FUNCTION_BLOCK FB_Status
VAR_INPUT
	eMode 	: E_Mode;
	fTime	: LREAL;
	bFault 	: BOOL;
END_VAR
VAR_OUTPUT
	eStatus : E_Status := E_Status.Checking;
END_VAR
VAR
	bRunning : BOOL;
END_VAR

IF fTime > 2.0 THEN
	bRunning := TRUE;
ELSE
	bRunning := FALSE;	
END_IF


CASE eStatus OF 
	E_Status.Checking:
		IF bFault THEN
			eStatus := E_Status.Fault;
		END_IF
		
		IF NOT(eMode = E_Mode.Off) AND NOT(bFault)THEN	
			eStatus := E_Status.Ready;
		END_IF
		
		IF eMode = E_Mode.Off THEN	
			eStatus := E_Status.Off;
		END_IF
		
	E_Status.Off:	
		IF NOT(eMode = E_Mode.Off) THEN	
			eStatus := E_Status.Checking;
		END_IF

	E_Status.Fault:
		IF NOT(bFault) THEN
			eStatus := E_Status.Checking;
		END_IF
	
	E_Status.Ready:
		IF G_Work.bStartButton AND NOT(eMode = E_Mode.Off) AND NOT(bFault) THEN
			eStatus := E_Status.Starting;
		END_IF	
		
		IF  eMode = E_Mode.Off OR bFault THEN
			eStatus := E_Status.Checking;
		END_IF	

	E_Status.Starting:
		IF bRunning THEN
			eStatus := E_Status.Running;
		END_IF 
		
		IF bFault OR eMode = E_Mode.Off  THEN
			eStatus := E_Status.Checking;
		END_IF
		
	
	E_Status.Running:
	
		IF G_Work.bStopButton THEN
			eStatus := E_Status.Stopping;
		END_IF
		
		IF NOT(bRunning) OR eMode = E_Mode.Off OR bFault THEN
			eStatus := E_Status.Checking;
		END_IF
	
	E_Status.Stopping:	
		IF NOT(bRunning) THEN
			eStatus := E_Status.Checking;
		END_IF
	
		IF eMode = E_Mode.Off OR bFault THEN
		eStatus := E_Status.Checking;
		END_IF	
	
ELSE 	
	eStatus := E_Status.Checking;
END_CASE

END_FUNCTION_BLOCK

(* stored: Version 1.1.0.1, ProductVersion 3.1.4024.13
   POU FB_Status: Id {26df518e-7453-4e6d-ac16-889885b93dbd}, SpecialFunc None *)
